# EPICS autosave request: softGlueApp/Db/softGlue_NPI_settings.req
file softGlue_SignalShow_settings.req P=$(P) H=$(H)
file softGlue_FPGAContent_NPI_settings.req P=$(P) H=$(H)
file softGlue_FPGAInt_settings.req P=$(P) H=$(H)
file softGlue_convenience_settings.req P=$(P) H=$(H)
